{attribute 'qualified_only'}
{attribute 'strict'}
TYPE E_ComponentMode :
(
	OFF 	:= 0,
	AUTO	:= 1,
	MANUAL	:= 2
);
END_TYPE

(* stored: Version 1.1.0.1, ProductVersion 3.1.4024.15
   EnumerationTextList E_ComponentMode: Id {4d22170d-f98a-46f8-95db-7e0072c23a48} *)
